(* CoDeSys 2.3 export: F_WRITE_TACK_VALVE_CFG.EXP *)

(* POU FUN/PARAMETERS/F_WRITE_TACK_VALVE_CFG, ST *)
FUNCTION F_WRITE_TACK_VALVE_CFG : BOOL
VAR_INPUT
	sHead : STRING;
	wSize   :DWORD;
	pBuffer :POINTER TO BYTE;
END_VAR
VAR_IN_OUT
	wPos     : DWORD;
	stConfig : ST_TACK_VALVE_CFG;
END_VAR
VAR
END_VAR
F_ADD_STRINGX3_TO_BUFFER( S1:= '$n#', S2:= sHead, S3:=' - Parameters:$n', wSize := wSize, pBuffer := pBuffer, wPos := wPos );

F_ADD_STRINGX4_TO_BUFFER( S1:= CONCAT(sHead, '_TimeMax'   ), S2:='$t', S3:= REAL_TO_STRING( stConfig.TimeMax  ), S4:='$n', wSize := wSize, pBuffer := pBuffer, wPos := wPos );

F_ADD_STRINGX4_TO_BUFFER( S1:= CONCAT(sHead, '_Hyst_HeelH' ), S2:='$t', S3:= REAL_TO_STRING( stConfig.Hyst_HeelH ), S4:='$n', wSize := wSize, pBuffer := pBuffer, wPos := wPos );
F_ADD_STRINGX4_TO_BUFFER( S1:= CONCAT(sHead, '_Hyst_HeelL' ), S2:='$t', S3:= REAL_TO_STRING( stConfig.Hyst_HeelL ), S4:='$n', wSize := wSize, pBuffer := pBuffer, wPos := wPos );
F_ADD_STRINGX4_TO_BUFFER( S1:= CONCAT(sHead, '_Hyst_Time'  ), S2:='$t', S3:= REAL_TO_STRING( stConfig.Hyst_Time  ), S4:='$n', wSize := wSize, pBuffer := pBuffer, wPos := wPos );
END_FUNCTION
